FUNCTION_BLOCK CROSSCOMM_SENDER_131AAE67C1B05F71B (* Service Interface Function Block Type *)
  (* Standard: 61499-2 *)
  (* Version 0.0, 9/22/2017, bababen, nxtControl GmbH, template *)
  PACKAGE Main;
  (* Compiler Cpp nxtControl builtin 1.0 *)
  {SET_ATTRIBUTE(Runtime.FBType.ImplementingType, Runtime.System#DYNGEN_CROSSCOMM_SENDER)}
  {SET_ATTRIBUTE(Configuration.GenericFBType.InterfaceParams, Runtime.System#<InterfaceList> <EventInputs> <Event Name="CNF"> <With Var="LiftRetractedCNF" /> <With Var="LiftExtendedCNF" /> </Event> </EventInputs> <InputVars> <VarDeclaration Name="LiftRetractedCNF" Type="BOOL" /> <VarDeclaration Name="LiftExtendedCNF" Type="BOOL" /> </InputVars> </InterfaceList>)}
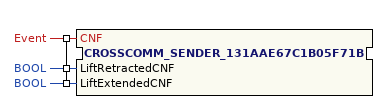
  EVENT_INPUT
    CNF WITH LiftRetractedCNF, LiftExtendedCNF;
  END_EVENT
  VAR_INPUT
    LiftRetractedCNF : BOOL;
    LiftExtendedCNF : BOOL;
  END_VAR
  EC_STATES
    START;
  END_STATES
END_FUNCTION_BLOCK
